(* IEC 61131-3 sources: Industry-PLC-LLM/data/PLCBEAD_repo/PLCBEAD_PLCEmbed-main/PLC-BEAD/Source/GEB/CADD, 1 file *)

(* ---- CADD.ST ---- *)
TYPE oscat_complex :
  STRUCT
	re : REAL;
	im : REAL;
  END_STRUCT;
END_TYPE

FUNCTION_BLOCK CADD_Block

	VAR_INPUT
		X :	oscat_complex;
		Y :	oscat_complex;
	END_VAR

	VAR_OUTPUT
		CADD :	oscat_complex;
	END_VAR

	CADD.re := X.re + Y.re;
	CADD.im := X.im + Y.im;

END_FUNCTION_BLOCK

PROGRAM program0
  VAR
    LocalVar0 : oscat_complex;
	LocalVaR1  : oscat_complex;
	LocalOUT  : oscat_complex;
	func_block : CADD_Block;
  END_VAR
	func_block.X  := LocalVar0;
	func_block.Y  := LocalVar0;
	func_block();
	LocalOUT := func_block.CADD;
END_PROGRAM
